Staubli VAL3: loadNextOne.pgx

program loadNextOne(string x_sName (dimensions=1))
begin
  prog_swap:libLoad(x_sName)
end
